# EPICS substitutions: pvNotepadApp/Db/ao_1.substitutions
#Substitutions for single substitution
file ao.template
{
    pattern { RECORD             }
            { $(HUTCH):NOTE:DOUBLE:01      }
}
